// SIMATIC S7-200 SMART project (STEP 7-Micro/WIN SMART), CPU ST40

SYMBOL_TABLE FACTORY IO
At_Entry         V0.0
At_Exit          V0.1
At_Load          V0.2
At_Unload        V0.3
Stacker_Middle_Limit V0.4
Stacker_Left_Limit V0.5
Stacker_Right_Limit V0.6
PUT_Button       V0.7
GET_Button       V1.0
EMT_Button       V1.1
RES_Button       V1.2
Moving_X         V1.3
Moving_Z         V1.4
FACTOR_IO_RESET  V1.5
SET              VD4
Stack            VW100
Stack_SZ         VW102
Entry_Conveyvor  Q0.0
Exit_Conveyor    Q0.1
Load_Conveyor    Q0.2
Unload_Conveyor  Q0.3
Lift             Q0.4
Stacker_Left     Q0.5
Stacker_Right    Q0.6
PUT_Light        Q0.7
GET_Light        Q1.0
EMT_Light        Q1.1
RES_Light        Q1.2
Target_Position  QD4
Position         QD8
Items_Count      QD12
END_SYMBOL_TABLE

SYMBOL_TABLE System Symbols
Always_On        SM0.0    // Always ON
First_Scan_On    SM0.1    // ON for the first scan cycle only
END_SYMBOL_TABLE

SYMBOL_TABLE MEM
M0               M0.0
M1               M0.1
M2               M0.2
M3               M0.3
M4               M0.4
M5               M0.5
M6               M0.6
M7               M0.7
M8               M1.0
M9               M1.1
M10              M1.2
M11              M1.3
M12              M1.4
M13              M1.5
M14              M1.6
M15              M1.7
Nxt              M31.7
END_SYMBOL_TABLE

ORGANIZATION_BLOCK MAIN:OB1
TITLE=Program Comments
VAR
SET_0:REAL;	// LD0  
Last_IN_I:INT;	// LW4 
Last_IN_DI:DINT;	// LD6 
END_VAR
BEGIN
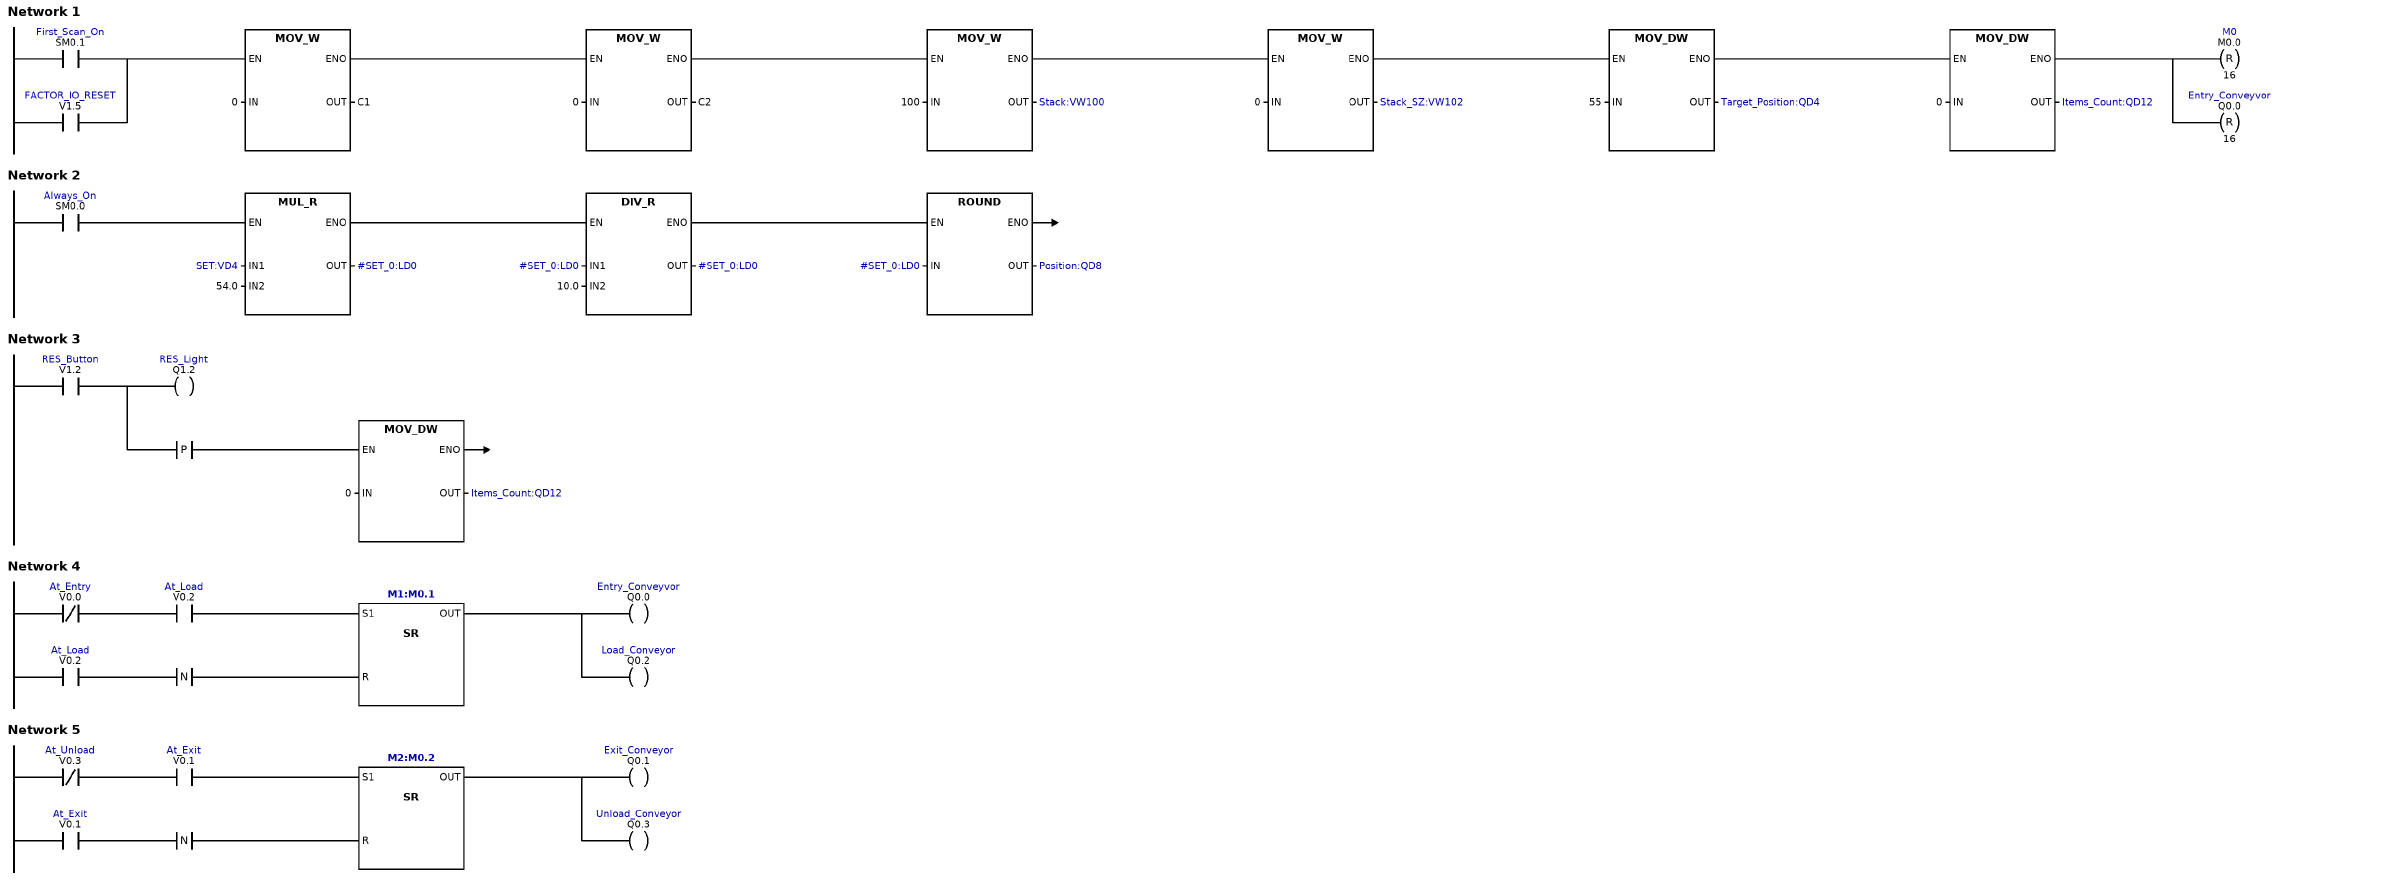
Network 1
LD     First_Scan_On:SM0.1
O      FACTOR_IO_RESET:V1.5
MOVW   0, C1
AENO
MOVW   0, C2
AENO
MOVW   100, Stack:VW100
AENO
MOVW   0, Stack_SZ:VW102
AENO
MOVD   55, Target_Position:QD4
AENO
MOVD   0, Items_Count:QD12
AENO
R      M0:M0.0, 16
R      Entry_Conveyvor:Q0.0, 16
Network 2
LD     Always_On:SM0.0
MOVR   SET:VD4, #SET_0:LD0
AENO
*R     54.0, #SET_0:LD0
AENO
/R     10.0, #SET_0:LD0
AENO
ROUND  #SET_0:LD0, Position:QD8
Network 3
LD     RES_Button:V1.2
=      RES_Light:Q1.2
EU
MOVD   0, Items_Count:QD12
Network 4
LDN    At_Entry:V0.0
A      At_Load:V0.2
LD     At_Load:V0.2
ED
NOT
A      M1:M0.1
OLD
=      M1:M0.1
=      Entry_Conveyvor:Q0.0
=      Load_Conveyor:Q0.2
Network 5
LDN    At_Unload:V0.3
A      At_Exit:V0.1
LD     At_Exit:V0.1
ED
NOT
A      M2:M0.2
OLD
=      M2:M0.2
=      Exit_Conveyor:Q0.1
=      Unload_Conveyor:Q0.3
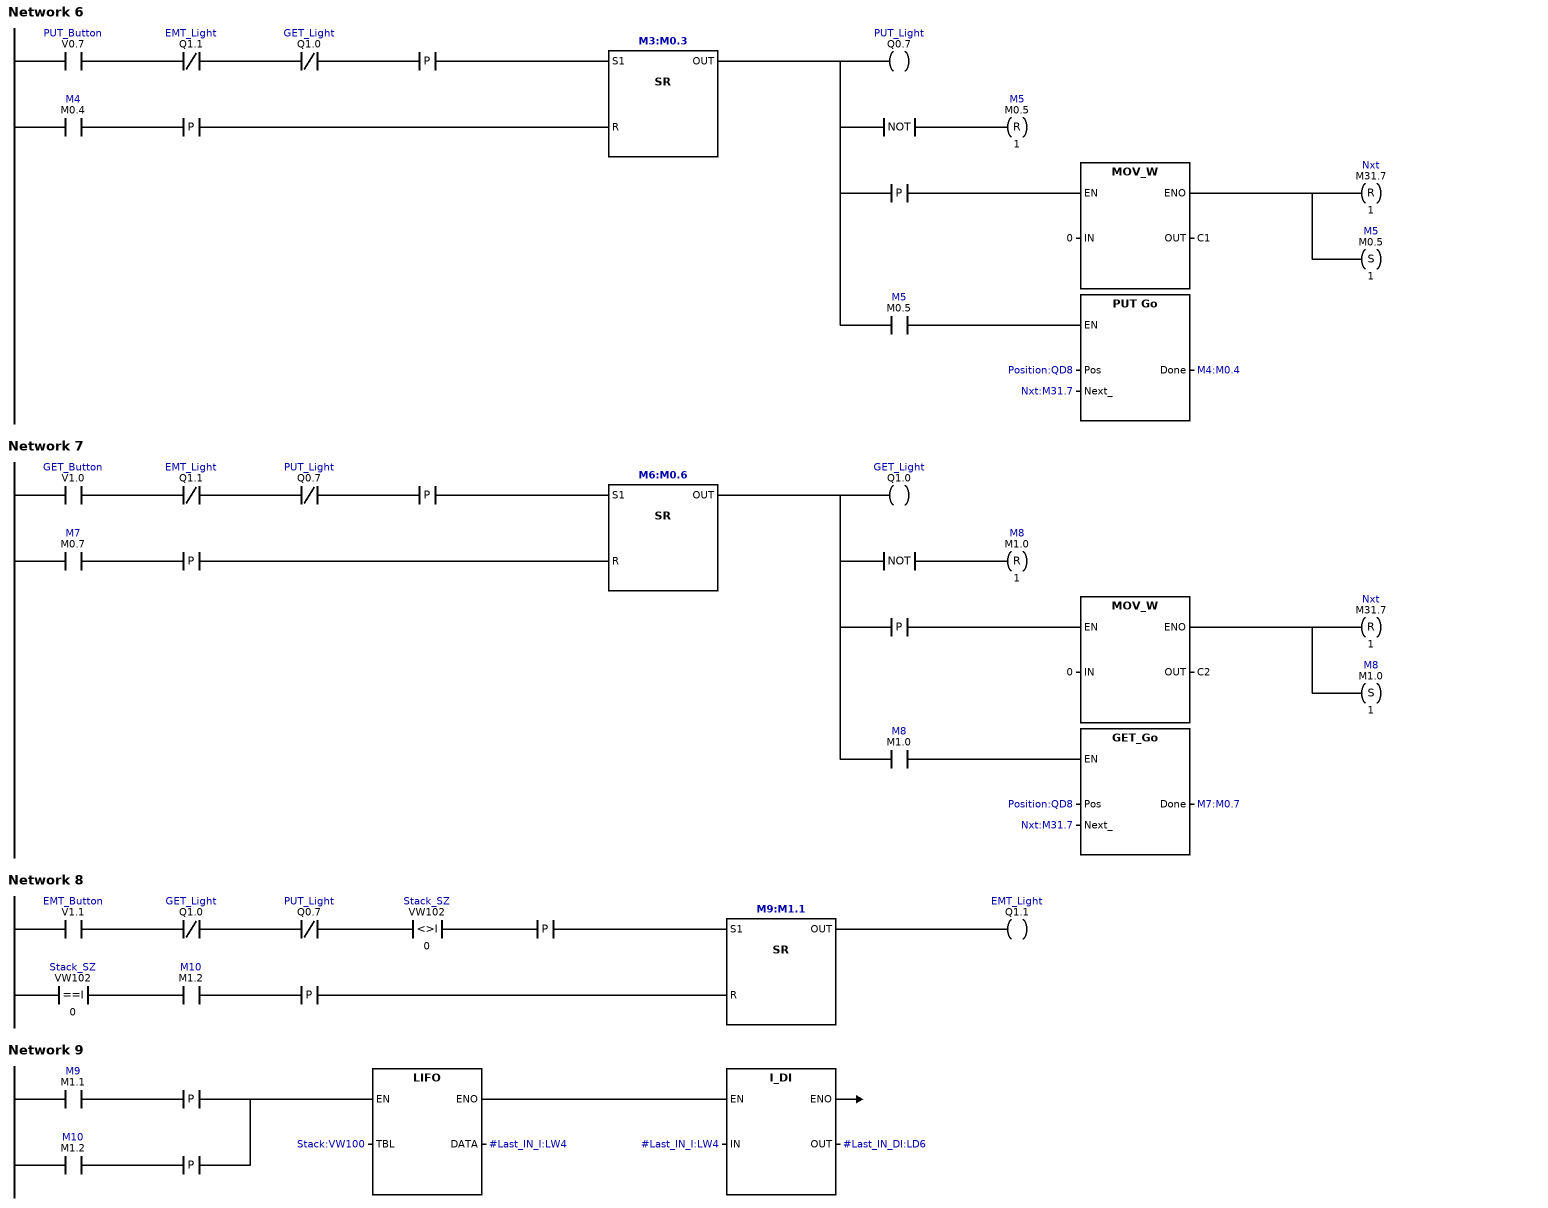
Network 6
LD     PUT_Button:V0.7
AN     EMT_Light:Q1.1
AN     GET_Light:Q1.0
EU
LD     M4:M0.4
EU
NOT
A      M3:M0.3
OLD
=      M3:M0.3
LPS
=      PUT_Light:Q0.7
NOT
R      M5:M0.5, 1
LRD
EU
MOVW   0, C1
AENO
R      Nxt:M31.7, 1
S      M5:M0.5, 1
LPP
A      M5:M0.5
CALL   PUT Go:SBR1, Position:QD8, Nxt:M31.7, M4:M0.4
Network 7
LD     GET_Button:V1.0
AN     EMT_Light:Q1.1
AN     PUT_Light:Q0.7
EU
LD     M7:M0.7
EU
NOT
A      M6:M0.6
OLD
=      M6:M0.6
LPS
=      GET_Light:Q1.0
NOT
R      M8:M1.0, 1
LRD
EU
MOVW   0, C2
AENO
R      Nxt:M31.7, 1
S      M8:M1.0, 1
LPP
A      M8:M1.0
CALL   GET_Go:SBR2, Position:QD8, Nxt:M31.7, M7:M0.7
Network 8
LD     EMT_Button:V1.1
AN     GET_Light:Q1.0
AN     PUT_Light:Q0.7
AW<>   Stack_SZ:VW102, 0
EU
LDW=   Stack_SZ:VW102, 0
A      M10:M1.2
EU
NOT
A      M9:M1.1
OLD
=      M9:M1.1
=      EMT_Light:Q1.1
Network 9
LD     M9:M1.1
EU
LD     M10:M1.2
EU
OLD
LIFO   Stack:VW100, #Last_IN_I:LW4
AENO
ITD    #Last_IN_I:LW4, #Last_IN_DI:LD6
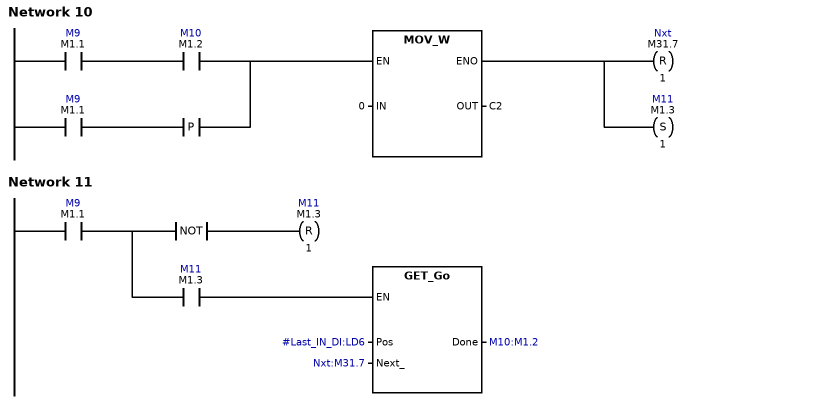
Network 10
LD     M9:M1.1
A      M10:M1.2
LD     M9:M1.1
EU
OLD
MOVW   0, C2
AENO
R      Nxt:M31.7, 1
S      M11:M1.3, 1
Network 11
LD     M9:M1.1
LPS
NOT
R      M11:M1.3, 1
LPP
A      M11:M1.3
CALL   GET_Go:SBR2, #Last_IN_DI:LD6, Nxt:M31.7, M10:M1.2
END_ORGANIZATION_BLOCK

SUBROUTINE_BLOCK Move:SBR0
TITLE=
VAR_INPUT
Pos:DWORD;	// LD0 
END_VAR
VAR_OUTPUT
Done:BOOL;	// L4.0 
END_VAR
BEGIN
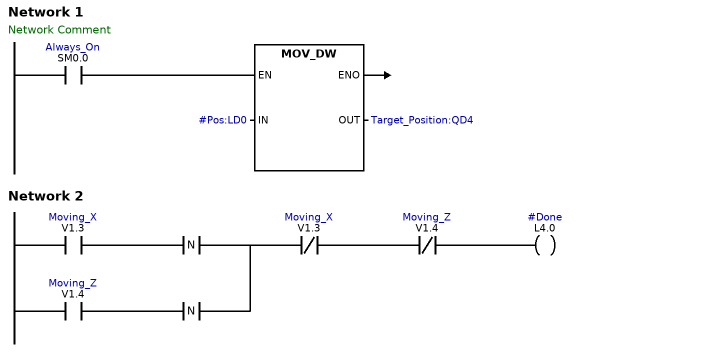
Network 1
// Network Comment
LD     Always_On:SM0.0
MOVD   #Pos:LD0, Target_Position:QD4
Network 2
LD     Moving_X:V1.3
ED
LD     Moving_Z:V1.4
ED
OLD
AN     Moving_X:V1.3
AN     Moving_Z:V1.4
=      #Done:L4.0
END_SUBROUTINE_BLOCK

SUBROUTINE_BLOCK PUT Go:SBR1
TITLE=
VAR_INPUT
Pos:DWORD;	// LD0 
END_VAR
VAR_IN_OUT
Next_:BOOL;	// L4.0 
END_VAR
VAR_OUTPUT
Done:BOOL;	// L4.1 
END_VAR
VAR
Pos_I:INT;	// LW5 
END_VAR
BEGIN
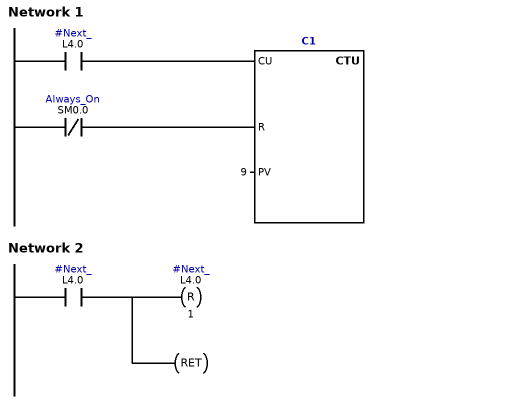
Network 1
LD     #Next_:L4.0
LDN    Always_On:SM0.0
CTU    C1, 9
Network 2
LD     #Next_:L4.0
R      #Next_:L4.0, 1
CRET
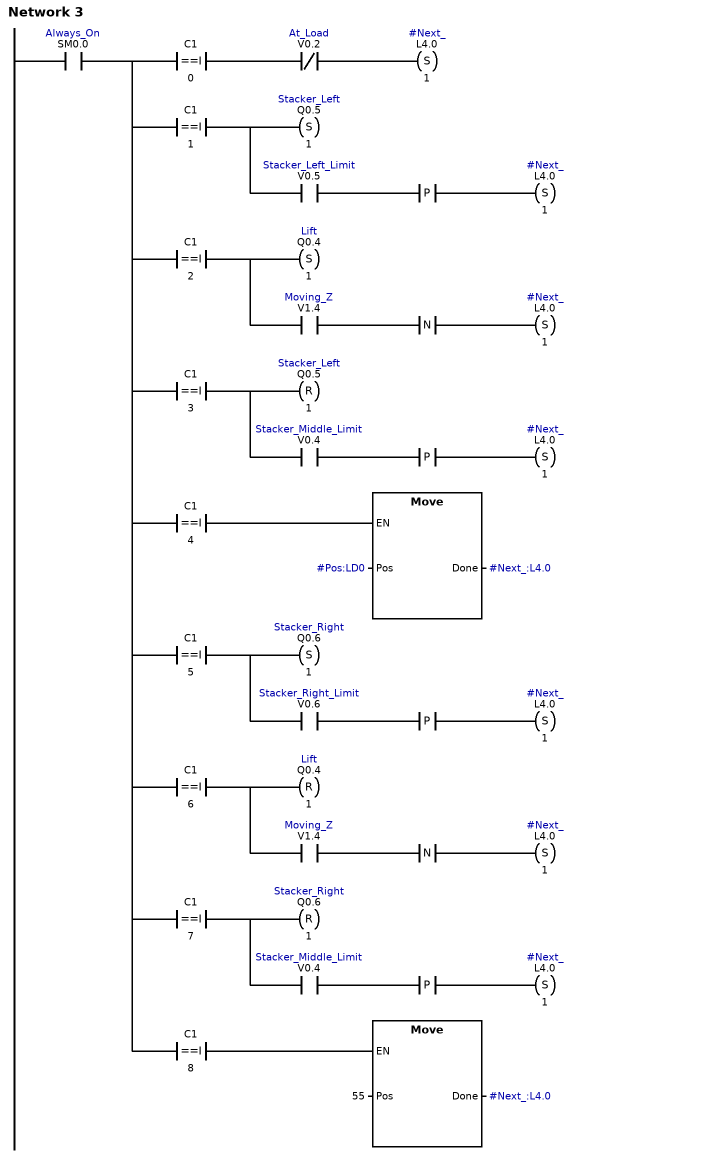
Network 3
LD     Always_On:SM0.0
LPS
AW=    C1, 0
AN     At_Load:V0.2
S      #Next_:L4.0, 1
LRD
AW=    C1, 1
S      Stacker_Left:Q0.5, 1
A      Stacker_Left_Limit:V0.5
EU
S      #Next_:L4.0, 1
LRD
AW=    C1, 2
S      Lift:Q0.4, 1
A      Moving_Z:V1.4
ED
S      #Next_:L4.0, 1
LRD
AW=    C1, 3
R      Stacker_Left:Q0.5, 1
A      Stacker_Middle_Limit:V0.4
EU
S      #Next_:L4.0, 1
LRD
AW=    C1, 4
CALL   Move:SBR0, #Pos:LD0, #Next_:L4.0
LRD
AW=    C1, 5
S      Stacker_Right:Q0.6, 1
A      Stacker_Right_Limit:V0.6
EU
S      #Next_:L4.0, 1
LRD
AW=    C1, 6
R      Lift:Q0.4, 1
A      Moving_Z:V1.4
ED
S      #Next_:L4.0, 1
LRD
AW=    C1, 7
R      Stacker_Right:Q0.6, 1
A      Stacker_Middle_Limit:V0.4
EU
S      #Next_:L4.0, 1
LPP
AW=    C1, 8
CALL   Move:SBR0, 55, #Next_:L4.0
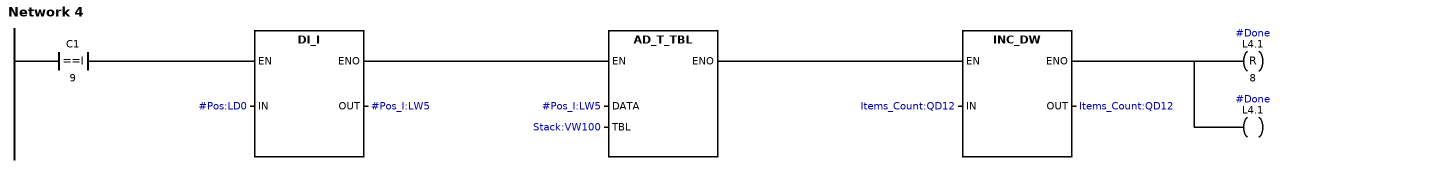
Network 4
LDW=   C1, 9
DTI    #Pos:LD0, #Pos_I:LW5
AENO
ATT    #Pos_I:LW5, Stack:VW100
AENO
INCD   Items_Count:QD12
AENO
R      #Done:L4.1, 8
=      #Done:L4.1
END_SUBROUTINE_BLOCK

SUBROUTINE_BLOCK GET_Go:SBR2
TITLE=
VAR_INPUT
Pos:DWORD;	// LD0 
END_VAR
VAR_IN_OUT
Next_:BOOL;	// L4.0 
END_VAR
VAR_OUTPUT
Done:BOOL;	// L4.1 
END_VAR
BEGIN
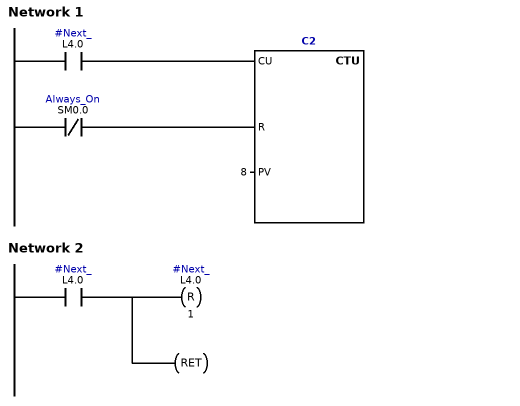
Network 1
LD     #Next_:L4.0
LDN    Always_On:SM0.0
CTU    C2, 8
Network 2
LD     #Next_:L4.0
R      #Next_:L4.0, 1
CRET
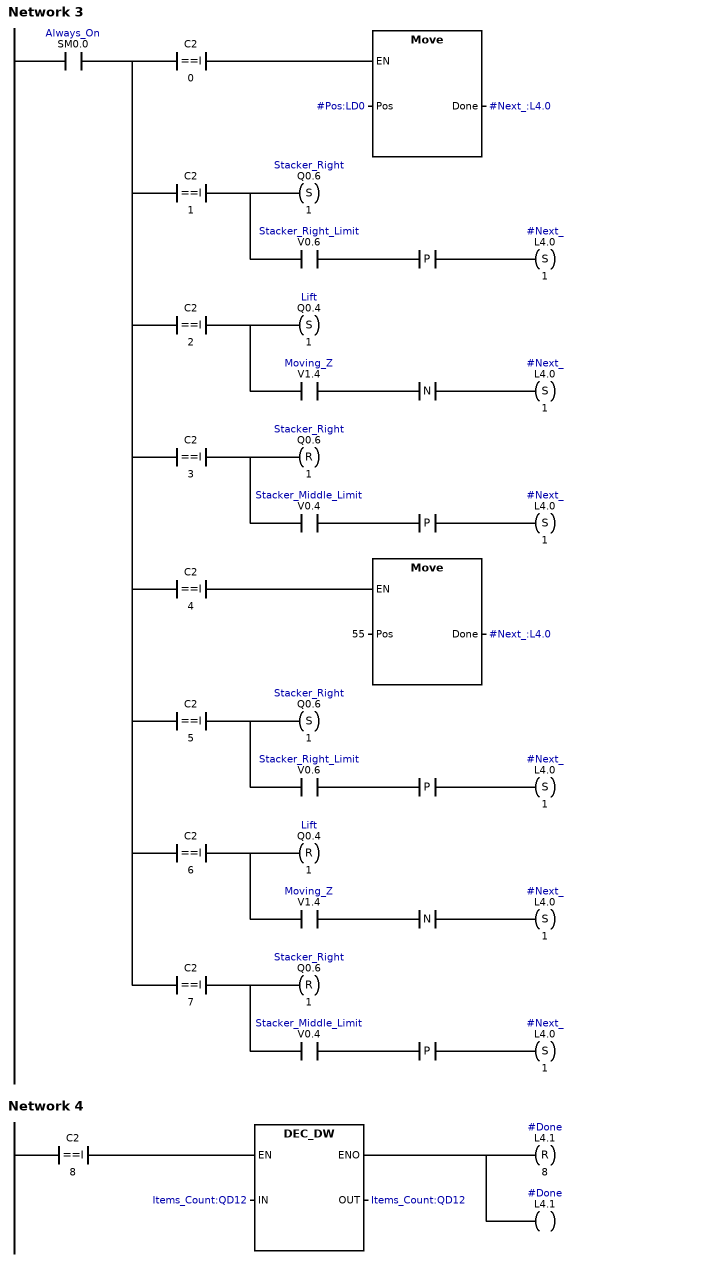
Network 3
LD     Always_On:SM0.0
LPS
AW=    C2, 0
CALL   Move:SBR0, #Pos:LD0, #Next_:L4.0
LRD
AW=    C2, 1
S      Stacker_Right:Q0.6, 1
A      Stacker_Right_Limit:V0.6
EU
S      #Next_:L4.0, 1
LRD
AW=    C2, 2
S      Lift:Q0.4, 1
A      Moving_Z:V1.4
ED
S      #Next_:L4.0, 1
LRD
AW=    C2, 3
R      Stacker_Right:Q0.6, 1
A      Stacker_Middle_Limit:V0.4
EU
S      #Next_:L4.0, 1
LRD
AW=    C2, 4
CALL   Move:SBR0, 55, #Next_:L4.0
LRD
AW=    C2, 5
S      Stacker_Right:Q0.6, 1
A      Stacker_Right_Limit:V0.6
EU
S      #Next_:L4.0, 1
LRD
AW=    C2, 6
R      Lift:Q0.4, 1
A      Moving_Z:V1.4
ED
S      #Next_:L4.0, 1
LPP
AW=    C2, 7
R      Stacker_Right:Q0.6, 1
A      Stacker_Middle_Limit:V0.4
EU
S      #Next_:L4.0, 1
Network 4
LDW=   C2, 8
DECD   Items_Count:QD12
AENO
R      #Done:L4.1, 8
=      #Done:L4.1
END_SUBROUTINE_BLOCK
